// TIA Portal V21 export
VAR_GLOBAL   // PLC tag table "K_ComunicazioneS7"
END_VAR
